// TIA Portal V20 export
TYPE "typeSequenceControlNode_transferPnPRight"
// stored: Namespace Unit1.Em5
   STRUCT
      jobs : "LAF_typeJobs";
      sequence : "LAF_typeSequence";
      selectJobStatus { S7_SetPoint := 'True'} : Array[0..10] of "LAF_typeJobStatus";
      "step" : "LER_typeStep";
      jobInterface : "Unit1.Em5.typeSequenceControlNodeJobInterface_transferPnPRight";
      homeCheck : "Unit1.Em5.typeSequenceControlNodeHomeCheck_transferPnPRight";
   END_STRUCT;
   // // "step".action1[101] : Step[101] : JOB[1] Condition
   // // "step".action1[110] : Step[110] : Transfer PP Right Clamp Open
   // // "step".action1[130] : Step[130] : Transfer PP Right Clamp Close
   // // "step".action1[160] : Step[160] : Transfer PP Right Y-Axis Wait Position
   // // "step".action1[170] : Step[170] : Transfer PP Right Z-Axis Wait Position
   // // "step".action1[180] : Step[180] : Transfer PP Right X-Axis Wait Position
   // // "step".action1[190] : Step[190] : JOB[1] Step End
   // // "step".action1[201] : Step[201] : JOB[2] Condition
   // // "step".action1[210] : Step[210] : Transfer PP Right X/Z-Axis Hipot & Thickness Pos
   // // "step".action1[230] : Step[230] : Transfer PP Right Y-Axis Hipot & Thickness Pos
   // // "step".action1[240] : Step[240] : Transfer PP Right Clamp Close
   // // "step".action1[280] : Step[280] : Transfer PP Right Y-Axis Wait Pos
   // // "step".action1[290] : Step[290] : JOB[2] Step End
   // // "step".action1[301] : Step[301] : JOB[3] Condition
   // // "step".action1[310] : Step[310] : Transfer PP Right X/Z-Axis Vision Pos
   // // "step".action1[330] : Step[330] : Transfer PP Right Y-Axis Vision Pos
   // // "step".action1[340] : Step[340] : Transfer PP Right [Lift Up Request] => Vision Check
   // // "step".action1[350] : Step[350] : Transfer PP Right Clamp Open
   // // "step".action1[380] : Step[380] : Transfer PP Right Y-Axis Wait Pos
   // // "step".action1[390] : Step[390] : JOB[3] Step End
   // // "step".action1[401] : Step[401] : JOB[4] Condition
   // // "step".action1[410] : Step[410] : Transfer PP Right X/Z-Axis Vision Pos
   // // "step".action1[430] : Step[430] : Transfer PP Right Y-Axis Vision Pos
   // // "step".action1[440] : Step[440] : Transfer PP Right Clamp Close
   // // "step".action1[480] : Step[480] : Transfer PP Right Y-Axis Wait Pos
   // // "step".action1[490] : Step[490] : JOB[4] Step End
   // // "step".action1[501] : Step[501] : JOB[5] Condition
   // // "step".action1[510] : Step[510] : Transfer PP Right X/Z-Axis Laser Mark Pos
   // // "step".action1[530] : Step[530] : Transfer PP Right Y-Axis Laser Mark Pos
   // // "step".action1[540] : Step[540] : Transfer PP Right [Lift Up Request] => Laser Mark
   // // "step".action1[550] : Step[550] : Transfer PP Right Clamp Open
   // // "step".action1[580] : Step[580] : Transfer PP Right Y-Axis Wait Pos
   // // "step".action1[590] : Step[590] : JOB[5] Step End
   // // "step".action1[601] : Step[601] : JOB[6] Condition
   // // "step".action1[602] : Step[602] : QR Read Start
   // // "step".action1[603] : Step[603] : QR Read Result
   // // "step".action1[604] : Step[604] : QR Read Start [NG]
   // // "step".action1[605] : Step[605] : QR Read Result [NG]
   // // "step".action1[610] : Step[610] : Transfer PP Right X/Z-Axis Laser Mark Pos
   // // "step".action1[630] : Step[630] : Transfer PP Right Y-Axis Laser Mark Pos
   // // "step".action1[640] : Step[640] : Transfer PP Right Clamp Close
   // // "step".action1[680] : Step[680] : Transfer PP Right Y-Axis Wait Pos
   // // "step".action1[690] : Step[690] : JOB[6] Step End
   // // "step".action1[701] : Step[701] : JOB[7] Condition
   // // "step".action1[710] : Step[710] : Transfer PP Right X/Z-Axis Laser Mark Pos
   // // "step".action1[730] : Step[730] : Transfer PP Right Y-Axis Laser Mark Pos
   // // "step".action1[740] : Step[740] : Transfer PP Right [Lift Up Request] => Laser Mark
   // // "step".action1[750] : Step[750] : Transfer PP Right Clamp Open
   // // "step".action1[780] : Step[780] : Transfer PP Right Y-Axis Wait Pos
   // // "step".action1[790] : Step[790] : JOB[7] Step End
   // // "step".action1[801] : Step[801] : JOB[8] Condition
   // // "step".action1[810] : Step[810] : Transfer PP Right X/Z-Axis Laser Mark Pos
   // // "step".action1[830] : Step[830] : Transfer PP Right Y-Axis Laser Mark Pos
   // // "step".action1[840] : Step[840] : Transfer PP Right Clamp Close
   // // "step".action1[880] : Step[880] : Transfer PP Right Y-Axis Wait Pos
   // // "step".action1[890] : Step[890] : JOB[8] Step End
   // // "step".action1[901] : Step[901] : JOB[9] Condition
   // // "step".action1[910] : Step[910] : Transfer PP Right X/Z-Axis Weight Check Pos
   // // "step".action1[930] : Step[930] : Transfer PP Right Y-Axis Weight Check Pos
   // // "step".action1[931] : Step[931] : Transfer PP Right Z-Axis Weight Check Pos
   // // "step".action1[940] : Step[940] : Transfer PP Right [Lift Up Request] => Weight Check
   // // "step".action1[950] : Step[950] : Transfer PP Right Clamp Open
   // // "step".action1[980] : Step[980] : Transfer PP Right Y-Axis Wait Pos
   // // "step".action1[981] : Step[981] : Transfer PP Right X/Z-Axis Wait Pos
   // // "step".action1[990] : Step[990] : JOB[9] Step End
   // // "step".transition1[101] : Step[101] : JOB[1] Condition
   // // "step".transition1[110] : Step[110] : Transfer PP Right Clamp Open
   // // "step".transition1[130] : Step[130] : Transfer PP Right Clamp Close
   // // "step".transition1[160] : Step[160] : Transfer PP Right Y-Axis Wait Position
   // // "step".transition1[170] : Step[170] : Transfer PP Right Z-Axis Wait Position
   // // "step".transition1[180] : Step[180] : Transfer PP Right X-Axis Wait Position
   // // "step".transition1[190] : Step[190] : JOB[1] Step End
   // // "step".transition1[201] : Step[201] : JOB[2] Condition
   // // "step".transition1[210] : Step[210] : Transfer PP Right X/Z-Axis Hipot & Thickness Pos
   // // "step".transition1[230] : Step[230] : Transfer PP Right Y-Axis Hipot & Thickness Pos
   // // "step".transition1[240] : Step[240] : Transfer PP Right Clamp Close
   // // "step".transition1[280] : Step[280] : Transfer PP Right Y-Axis Wait Pos
   // // "step".transition1[290] : Step[290] : JOB[2] Step End
   // // "step".transition1[301] : Step[301] : JOB[3] Condition
   // // "step".transition1[310] : Step[310] : Transfer PP Right X/Z-Axis Vision Pos
   // // "step".transition1[330] : Step[330] : Transfer PP Right Y-Axis Vision Pos
   // // "step".transition1[340] : Step[340] : Transfer PP Right [Lift Up Request] => Vision Check
   // // "step".transition1[350] : Step[350] : Transfer PP Right Clamp Open
   // // "step".transition1[380] : Step[380] : Transfer PP Right Y-Axis Wait Pos
   // // "step".transition1[390] : Step[390] : JOB[3] Step End
   // // "step".transition1[401] : Step[401] : JOB[4] Condition
   // // "step".transition1[410] : Step[410] : Transfer PP Right X/Z-Axis Vision Pos
   // // "step".transition1[430] : Step[430] : Transfer PP Right Y-Axis Vision Pos
   // // "step".transition1[440] : Step[440] : Transfer PP Right Clamp Close
   // // "step".transition1[480] : Step[480] : Transfer PP Right Y-Axis Wait Pos
   // // "step".transition1[490] : Step[490] : JOB[4] Step End
   // // "step".transition1[501] : Step[501] : JOB[5] Condition
   // // "step".transition1[510] : Step[510] : Transfer PP Right X/Z-Axis Laser Mark Pos
   // // "step".transition1[530] : Step[530] : Transfer PP Right Y-Axis Laser Mark Pos
   // // "step".transition1[540] : Step[540] : Transfer PP Right [Lift Up Request] => Laser Mark
   // // "step".transition1[550] : Step[550] : Transfer PP Right Clamp Open
   // // "step".transition1[580] : Step[580] : Transfer PP Right Y-Axis Wait Pos
   // // "step".transition1[590] : Step[590] : JOB[5] Step End
   // // "step".transition1[601] : Step[601] : JOB[6] Condition
   // // "step".transition1[602] : Step[602] : QR Read Start
   // // "step".transition1[603] : Step[603] : QR Read Result
   // // "step".transition1[604] : Step[604] : QR Read Start [NG]
   // // "step".transition1[605] : Step[605] : QR Read Result [NG]
   // // "step".transition1[610] : Step[610] : Transfer PP Right X/Z-Axis Laser Mark Pos
   // // "step".transition1[630] : Step[630] : Transfer PP Right Y-Axis Laser Mark Pos
   // // "step".transition1[640] : Step[640] : Transfer PP Right Clamp Close
   // // "step".transition1[680] : Step[680] : Transfer PP Right Y-Axis Wait Pos
   // // "step".transition1[690] : Step[690] : JOB[6] Step End
   // // "step".transition1[701] : Step[701] : JOB[7] Condition
   // // "step".transition1[710] : Step[710] : Transfer PP Right X/Z-Axis Laser Mark Pos
   // // "step".transition1[730] : Step[730] : Transfer PP Right Y-Axis Laser Mark Pos
   // // "step".transition1[740] : Step[740] : Transfer PP Right [Lift Up Request] => Laser Mark
   // // "step".transition1[750] : Step[750] : Transfer PP Right Clamp Open
   // // "step".transition1[780] : Step[780] : Transfer PP Right Y-Axis Wait Pos
   // // "step".transition1[790] : Step[790] : JOB[7] Step End
   // // "step".transition1[801] : Step[801] : JOB[8] Condition
   // // "step".transition1[810] : Step[810] : Transfer PP Right X/Z-Axis Laser Mark Pos
   // // "step".transition1[830] : Step[830] : Transfer PP Right Y-Axis Laser Mark Pos
   // // "step".transition1[840] : Step[840] : Transfer PP Right Clamp Close
   // // "step".transition1[880] : Step[880] : Transfer PP Right Y-Axis Wait Pos
   // // "step".transition1[890] : Step[890] : JOB[8] Step End
   // // "step".transition1[901] : Step[901] : JOB[9] Condition
   // // "step".transition1[910] : Step[910] : Transfer PP Right X/Z-Axis Weight Check Pos
   // // "step".transition1[930] : Step[930] : Transfer PP Right Y-Axis Weight Check Pos
   // // "step".transition1[931] : Step[931] : Transfer PP Right Z-Axis Weight Check Pos
   // // "step".transition1[940] : Step[940] : Transfer PP Right [Lift Up Request] => Weight Check
   // // "step".transition1[950] : Step[950] : Transfer PP Right Clamp Open
   // // "step".transition1[980] : Step[980] : Transfer PP Right Y-Axis Wait Pos
   // // "step".transition1[981] : Step[981] : Transfer PP Right X/Z-Axis Wait Pos
   // // "step".transition1[990] : Step[990] : JOB[9] Step End
END_TYPE
